// TIA Portal project "banc de percage" (V16)

(* hardware
DEVICE "Station S7-1200_1"  S7-1200 Station
   slot 0: "Châssis_0"  S7-1200 Rack  Rack  V1.0
   slot 1: "PLC_1"  CPU 1214C DC/DC/DC  6ES7 214-1AG31-0XB0  V3.0
*)

// ===== PLC "PLC_1"  CPU 1214C DC/DC/DC =====

VAR_GLOBAL   // PLC tag table "Table de variables standard"
   "S1" AT %I0.0 : Bool;
   "AU" AT %I0.1 : Bool;
   "DCA" AT %I0.2 : Bool;
   "FCA" AT %I0.3 : Bool;
   "DCB" AT %I0.4 : Bool;
   "FCB" AT %I0.5 : Bool;
   "FCC" AT %I0.6 : Bool;
   "PP" AT %I0.7 : Bool;
   "SWC" AT %I1.0 : Bool;
   "A12" AT %Q0.1 : Bool;
   "A14" AT %Q0.2 : Bool;
   "B12" AT %Q0.3 : Bool;
   "B14" AT %Q0.4 : Bool;
   "D12" AT %Q0.5 : Bool;
   "KM1" AT %Q0.6 : Bool;
   "H1" AT %Q0.7 : Bool;
   "H2" AT %Q1.0 : Bool;
   "Mot etape" AT %MW20 : Int;
   "Clock_Byte" AT %MB0 : Byte;
   "Clock_10Hz" AT %M0.0 : Bool;
   "Clock_5Hz" AT %M0.1 : Bool;
   "Clock_2.5Hz" AT %M0.2 : Bool;
   "Clock_2Hz" AT %M0.3 : Bool;
   "Clock_1.25Hz" AT %M0.4 : Bool;
   "Clock_1Hz" AT %M0.5 : Bool;
   "Clock_0.625Hz" AT %M0.6 : Bool;
   "Clock_0.5Hz" AT %M0.7 : Bool;
   "RAU" AT %I1.1 : Bool;
   "H3" AT %Q1.1 : Bool;
   "Reset" AT %E1.2 : Bool;
   "C12" AT %Q0.0 : Bool;
END_VAR

// folder: System blocks/Program resources

DATA_BLOCK "IEC_Timer_0_DB_1"   // DB2
{ S7_Optimized_Access := 'TRUE' }
AUTHOR : Simatic
FAMILY : IEC
NAME : IEC_TMR
VERSION : 1.0
// stored: InstanceOfName IEC_TIMER
"IEC_TIMER"
BEGIN
END_DATA_BLOCK

DATA_BLOCK "IEC_Timer_0_DB_2"   // DB3
{ S7_Optimized_Access := 'TRUE' }
AUTHOR : Simatic
FAMILY : IEC
NAME : IEC_TMR
VERSION : 1.0
// stored: InstanceOfName IEC_TIMER
"IEC_TIMER"
BEGIN
END_DATA_BLOCK

DATA_BLOCK "IEC_Timer_0_DB_3"   // DB4
{ S7_Optimized_Access := 'TRUE' }
AUTHOR : Simatic
FAMILY : IEC
NAME : IEC_TMR
VERSION : 1.0
// stored: InstanceOfName IEC_TIMER
"IEC_TIMER"
BEGIN
END_DATA_BLOCK

// folder: (top level)

FUNCTION "Transition" : Void   // FC1, LAD
{ S7_Optimized_Access := 'TRUE' }
VERSION : 0.1
   VAR_TEMP   // added for the SCL form of the ladder/FBD networks
      _w1 : Bool;
   END_VAR
BEGIN

REGION Network 1
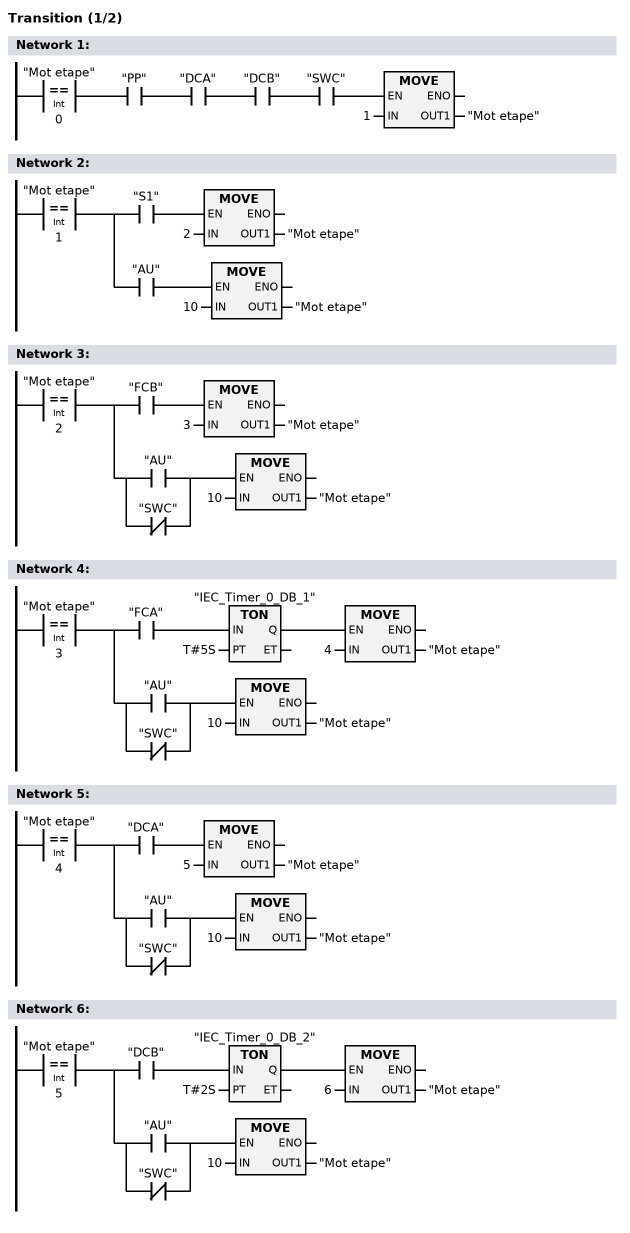
   RUNG wire#powerrail
      { S7_Templates := "SrcType := Int" } EQ_Contact(in1 := "Mot etape", in2 := 0)
      Contact( "PP" )
      Contact( "DCA" )
      Contact( "DCB" )
      Contact( "SWC" )
      { S7_GenerateENO := "TRUE" } Move(in := 1, out1 => "Mot etape")
   END_RUNG
   // the same network as SCL:
   IF ("Mot etape" = 0) AND "PP" AND "DCA" AND "DCB" AND "SWC" THEN "Mot etape" := 1; END_IF;
END_REGION

REGION Network 2
   RUNG wire#powerrail
      { S7_Templates := "SrcType := Int" } EQ_Contact(in1 := "Mot etape", in2 := 1)
      wire#w1
      Contact( "S1" )
      { S7_GenerateENO := "TRUE" } Move(in := 2, out1 => "Mot etape")
   END_RUNG
   RUNG wire#w1
      Contact( "AU" )
      { S7_GenerateENO := "TRUE" } Move(in := 10, out1 => "Mot etape")
   END_RUNG
   // the same network as SCL:
   #_w1 := "Mot etape" = 1;
   IF #_w1 AND "S1" THEN "Mot etape" := 2; END_IF;
   IF #_w1 AND "AU" THEN "Mot etape" := 10; END_IF;
END_REGION

REGION Network 3
   RUNG wire#powerrail
      { S7_Templates := "SrcType := Int" } EQ_Contact(in1 := "Mot etape", in2 := 2)
      wire#w1
      Contact( "FCB" )
      { S7_GenerateENO := "TRUE" } Move(in := 3, out1 => "Mot etape")
   END_RUNG
   RUNG wire#w1
      Contact( "AU" )
      wire#w2
      { S7_GenerateENO := "TRUE" } Move(in := 10, out1 => "Mot etape")
   END_RUNG
   RUNG wire#w1
      I_Contact( "SWC" )
   END_RUNG wire#w2
   // the same network as SCL:
   #_w1 := "Mot etape" = 2;
   IF #_w1 AND "FCB" THEN "Mot etape" := 3; END_IF;
   IF #_w1 AND ("AU" OR NOT "SWC") THEN "Mot etape" := 10; END_IF;
END_REGION

REGION Network 4
   #_w1 := "Mot etape" = 3;
   "IEC_Timer_0_DB_1".TON(IN := #_w1 AND "FCA", PT := T#5S);
   IF "IEC_Timer_0_DB_1".Q THEN "Mot etape" := 4; END_IF;
   IF #_w1 AND ("AU" OR NOT "SWC") THEN "Mot etape" := 10; END_IF;
END_REGION

REGION Network 5
   RUNG wire#powerrail
      { S7_Templates := "SrcType := Int" } EQ_Contact(in1 := "Mot etape", in2 := 4)
      wire#w1
      Contact( "DCA" )
      { S7_GenerateENO := "TRUE" } Move(in := 5, out1 => "Mot etape")
   END_RUNG
   RUNG wire#w1
      Contact( "AU" )
      wire#w2
      { S7_GenerateENO := "TRUE" } Move(in := 10, out1 => "Mot etape")
   END_RUNG
   RUNG wire#w1
      I_Contact( "SWC" )
   END_RUNG wire#w2
   // the same network as SCL:
   #_w1 := "Mot etape" = 4;
   IF #_w1 AND "DCA" THEN "Mot etape" := 5; END_IF;
   IF #_w1 AND ("AU" OR NOT "SWC") THEN "Mot etape" := 10; END_IF;
END_REGION

REGION Network 6
   #_w1 := "Mot etape" = 5;
   "IEC_Timer_0_DB_2".TON(IN := #_w1 AND "DCB", PT := T#2S);
   IF "IEC_Timer_0_DB_2".Q THEN "Mot etape" := 6; END_IF;
   IF #_w1 AND ("AU" OR NOT "SWC") THEN "Mot etape" := 10; END_IF;
END_REGION

REGION Network 7
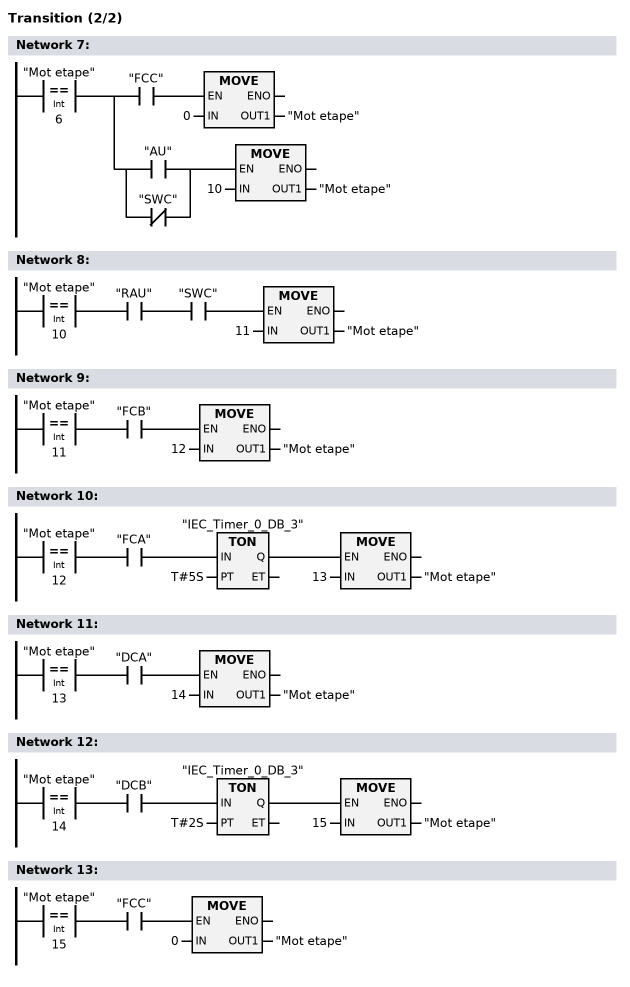
   RUNG wire#powerrail
      { S7_Templates := "SrcType := Int" } EQ_Contact(in1 := "Mot etape", in2 := 6)
      wire#w1
      Contact( "FCC" )
      { S7_GenerateENO := "TRUE" } Move(in := 0, out1 => "Mot etape")
   END_RUNG
   RUNG wire#w1
      Contact( "AU" )
      wire#w2
      { S7_GenerateENO := "TRUE" } Move(in := 10, out1 => "Mot etape")
   END_RUNG
   RUNG wire#w1
      I_Contact( "SWC" )
   END_RUNG wire#w2
   // the same network as SCL:
   #_w1 := "Mot etape" = 6;
   IF #_w1 AND "FCC" THEN "Mot etape" := 0; END_IF;
   IF #_w1 AND ("AU" OR NOT "SWC") THEN "Mot etape" := 10; END_IF;
END_REGION

REGION Network 8
   RUNG wire#powerrail
      { S7_Templates := "SrcType := Int" } EQ_Contact(in1 := "Mot etape", in2 := 10)
      Contact( "RAU" )
      Contact( "SWC" )
      { S7_GenerateENO := "TRUE" } Move(in := 11, out1 => "Mot etape")
   END_RUNG
   // the same network as SCL:
   IF ("Mot etape" = 10) AND "RAU" AND "SWC" THEN "Mot etape" := 11; END_IF;
END_REGION

REGION Network 9
   RUNG wire#powerrail
      { S7_Templates := "SrcType := Int" } EQ_Contact(in1 := "Mot etape", in2 := 11)
      Contact( "FCB" )
      { S7_GenerateENO := "TRUE" } Move(in := 12, out1 => "Mot etape")
   END_RUNG
   // the same network as SCL:
   IF ("Mot etape" = 11) AND "FCB" THEN "Mot etape" := 12; END_IF;
END_REGION

REGION Network 10
   "IEC_Timer_0_DB_3".TON(IN := ("Mot etape" = 12) AND "FCA", PT := T#5S);
   IF "IEC_Timer_0_DB_3".Q THEN "Mot etape" := 13; END_IF;
END_REGION

REGION Network 11
   RUNG wire#powerrail
      { S7_Templates := "SrcType := Int" } EQ_Contact(in1 := "Mot etape", in2 := 13)
      Contact( "DCA" )
      { S7_GenerateENO := "TRUE" } Move(in := 14, out1 => "Mot etape")
   END_RUNG
   // the same network as SCL:
   IF ("Mot etape" = 13) AND "DCA" THEN "Mot etape" := 14; END_IF;
END_REGION

REGION Network 12
   "IEC_Timer_0_DB_3".TON(IN := ("Mot etape" = 14) AND "DCB", PT := T#2S);
   IF "IEC_Timer_0_DB_3".Q THEN "Mot etape" := 15; END_IF;
END_REGION

REGION Network 13
   RUNG wire#powerrail
      { S7_Templates := "SrcType := Int" } EQ_Contact(in1 := "Mot etape", in2 := 15)
      Contact( "FCC" )
      { S7_GenerateENO := "TRUE" } Move(in := 0, out1 => "Mot etape")
   END_RUNG
   // the same network as SCL:
   IF ("Mot etape" = 15) AND "FCC" THEN "Mot etape" := 0; END_IF;
END_REGION
END_FUNCTION

FUNCTION "Sortie" : Void   // FC2, LAD
{ S7_Optimized_Access := 'TRUE' }
VERSION : 0.1
BEGIN

REGION Network 1
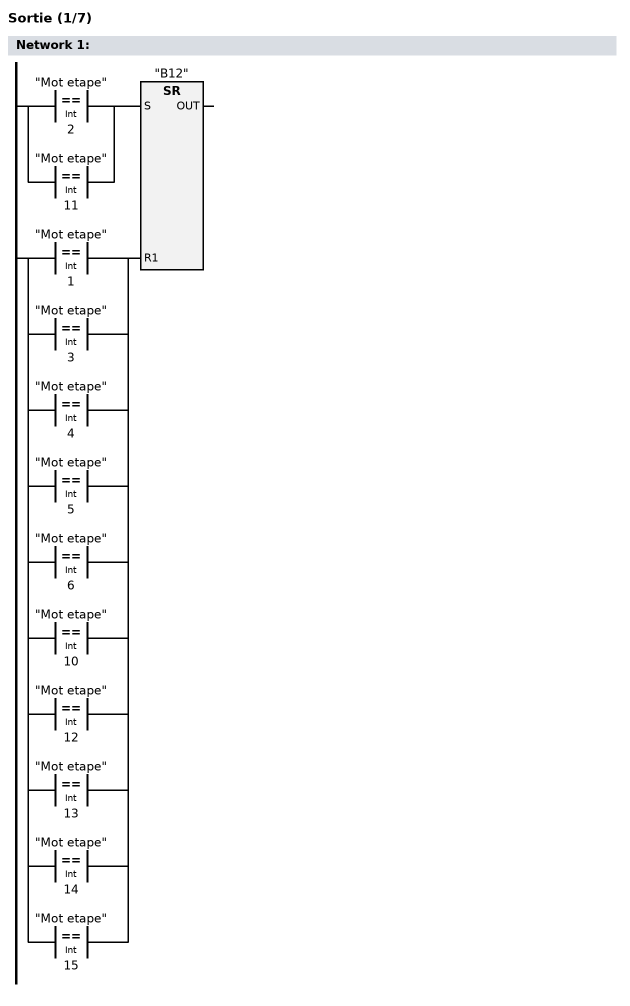
   RUNG wire#powerrail
      { S7_Templates := "SrcType := Int" } EQ_Contact(in1 := "Mot etape", in2 := 2)
      wire#w1
      S_SR(operand := "B12", r1 := wire#w2)
   END_RUNG
   RUNG wire#powerrail
      { S7_Templates := "SrcType := Int" } EQ_Contact(in1 := "Mot etape", in2 := 11)
   END_RUNG wire#w1
   RUNG wire#powerrail
      { S7_Templates := "SrcType := Int" } EQ_Contact(in1 := "Mot etape", in2 := 1)
   END_RUNG wire#w2
   RUNG wire#powerrail
      { S7_Templates := "SrcType := Int" } EQ_Contact(in1 := "Mot etape", in2 := 3)
   END_RUNG wire#w2
   RUNG wire#powerrail
      { S7_Templates := "SrcType := Int" } EQ_Contact(in1 := "Mot etape", in2 := 4)
   END_RUNG wire#w2
   RUNG wire#powerrail
      { S7_Templates := "SrcType := Int" } EQ_Contact(in1 := "Mot etape", in2 := 5)
   END_RUNG wire#w2
   RUNG wire#powerrail
      { S7_Templates := "SrcType := Int" } EQ_Contact(in1 := "Mot etape", in2 := 6)
   END_RUNG wire#w2
   RUNG wire#powerrail
      { S7_Templates := "SrcType := Int" } EQ_Contact(in1 := "Mot etape", in2 := 10)
   END_RUNG wire#w2
   RUNG wire#powerrail
      { S7_Templates := "SrcType := Int" } EQ_Contact(in1 := "Mot etape", in2 := 12)
   END_RUNG wire#w2
   RUNG wire#powerrail
      { S7_Templates := "SrcType := Int" } EQ_Contact(in1 := "Mot etape", in2 := 13)
   END_RUNG wire#w2
   RUNG wire#powerrail
      { S7_Templates := "SrcType := Int" } EQ_Contact(in1 := "Mot etape", in2 := 14)
   END_RUNG wire#w2
   RUNG wire#powerrail
      { S7_Templates := "SrcType := Int" } EQ_Contact(in1 := "Mot etape", in2 := 15)
   END_RUNG wire#w2
   // the same network as SCL:
   IF ("Mot etape" = 2) OR ("Mot etape" = 11) THEN
       "B12" := TRUE;   // SR flip-flop
   END_IF;
   IF ("Mot etape" = 1) OR ("Mot etape" = 3) OR ("Mot etape" = 4) OR ("Mot etape" = 5) OR ("Mot etape" = 6) OR ("Mot etape" = 10) OR ("Mot etape" = 12) OR ("Mot etape" = 13) OR ("Mot etape" = 14) OR ("Mot etape" = 15) THEN
       "B12" := FALSE;
   END_IF;
END_REGION

REGION Network 2
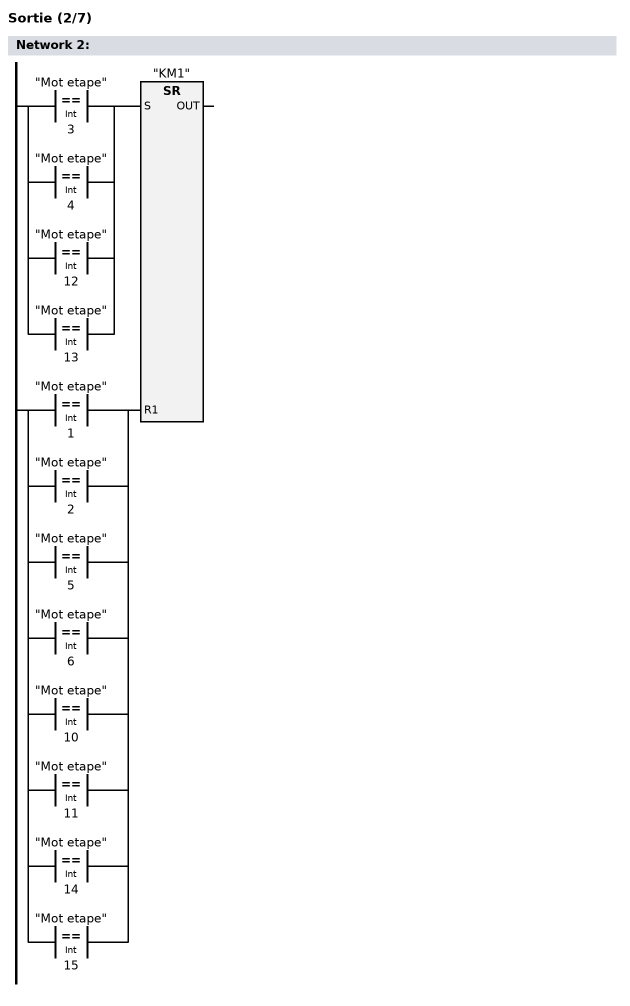
   RUNG wire#powerrail
      { S7_Templates := "SrcType := Int" } EQ_Contact(in1 := "Mot etape", in2 := 3)
      wire#w1
      S_SR(operand := "KM1", r1 := wire#w2)
   END_RUNG
   RUNG wire#powerrail
      { S7_Templates := "SrcType := Int" } EQ_Contact(in1 := "Mot etape", in2 := 4)
   END_RUNG wire#w1
   RUNG wire#powerrail
      { S7_Templates := "SrcType := Int" } EQ_Contact(in1 := "Mot etape", in2 := 12)
   END_RUNG wire#w1
   RUNG wire#powerrail
      { S7_Templates := "SrcType := Int" } EQ_Contact(in1 := "Mot etape", in2 := 13)
   END_RUNG wire#w1
   RUNG wire#powerrail
      { S7_Templates := "SrcType := Int" } EQ_Contact(in1 := "Mot etape", in2 := 1)
   END_RUNG wire#w2
   RUNG wire#powerrail
      { S7_Templates := "SrcType := Int" } EQ_Contact(in1 := "Mot etape", in2 := 2)
   END_RUNG wire#w2
   RUNG wire#powerrail
      { S7_Templates := "SrcType := Int" } EQ_Contact(in1 := "Mot etape", in2 := 5)
   END_RUNG wire#w2
   RUNG wire#powerrail
      { S7_Templates := "SrcType := Int" } EQ_Contact(in1 := "Mot etape", in2 := 6)
   END_RUNG wire#w2
   RUNG wire#powerrail
      { S7_Templates := "SrcType := Int" } EQ_Contact(in1 := "Mot etape", in2 := 10)
   END_RUNG wire#w2
   RUNG wire#powerrail
      { S7_Templates := "SrcType := Int" } EQ_Contact(in1 := "Mot etape", in2 := 11)
   END_RUNG wire#w2
   RUNG wire#powerrail
      { S7_Templates := "SrcType := Int" } EQ_Contact(in1 := "Mot etape", in2 := 14)
   END_RUNG wire#w2
   RUNG wire#powerrail
      { S7_Templates := "SrcType := Int" } EQ_Contact(in1 := "Mot etape", in2 := 15)
   END_RUNG wire#w2
   // the same network as SCL:
   IF ("Mot etape" = 3) OR ("Mot etape" = 4) OR ("Mot etape" = 12) OR ("Mot etape" = 13) THEN
       "KM1" := TRUE;   // SR flip-flop
   END_IF;
   IF ("Mot etape" = 1) OR ("Mot etape" = 2) OR ("Mot etape" = 5) OR ("Mot etape" = 6) OR ("Mot etape" = 10) OR ("Mot etape" = 11) OR ("Mot etape" = 14) OR ("Mot etape" = 15) THEN
       "KM1" := FALSE;
   END_IF;
END_REGION

REGION Network 3
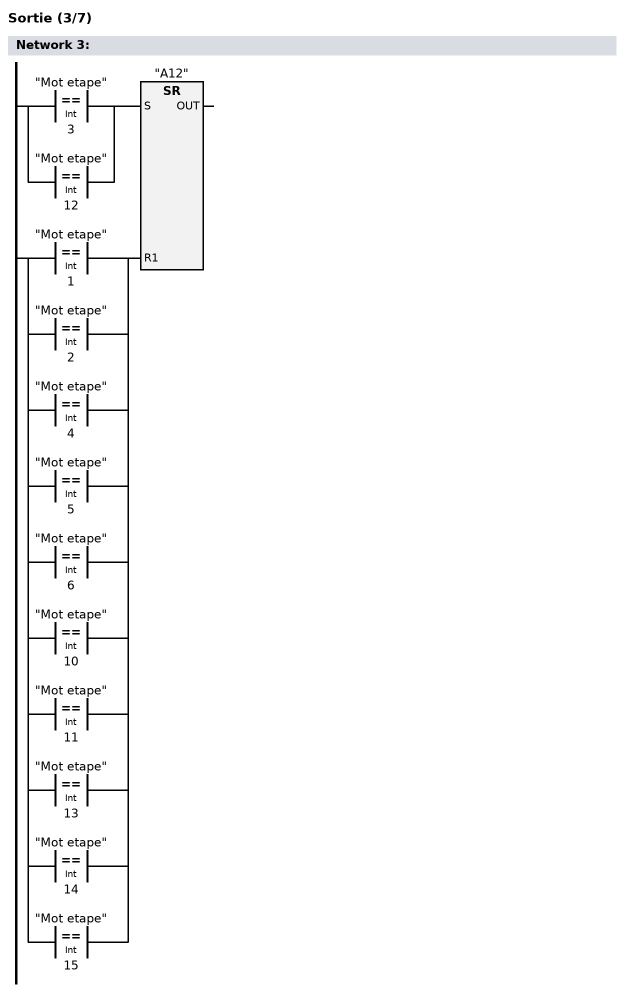
   RUNG wire#powerrail
      { S7_Templates := "SrcType := Int" } EQ_Contact(in1 := "Mot etape", in2 := 3)
      wire#w1
      S_SR(operand := "A12", r1 := wire#w2)
   END_RUNG
   RUNG wire#powerrail
      { S7_Templates := "SrcType := Int" } EQ_Contact(in1 := "Mot etape", in2 := 12)
   END_RUNG wire#w1
   RUNG wire#powerrail
      { S7_Templates := "SrcType := Int" } EQ_Contact(in1 := "Mot etape", in2 := 1)
   END_RUNG wire#w2
   RUNG wire#powerrail
      { S7_Templates := "SrcType := Int" } EQ_Contact(in1 := "Mot etape", in2 := 2)
   END_RUNG wire#w2
   RUNG wire#powerrail
      { S7_Templates := "SrcType := Int" } EQ_Contact(in1 := "Mot etape", in2 := 4)
   END_RUNG wire#w2
   RUNG wire#powerrail
      { S7_Templates := "SrcType := Int" } EQ_Contact(in1 := "Mot etape", in2 := 5)
   END_RUNG wire#w2
   RUNG wire#powerrail
      { S7_Templates := "SrcType := Int" } EQ_Contact(in1 := "Mot etape", in2 := 6)
   END_RUNG wire#w2
   RUNG wire#powerrail
      { S7_Templates := "SrcType := Int" } EQ_Contact(in1 := "Mot etape", in2 := 10)
   END_RUNG wire#w2
   RUNG wire#powerrail
      { S7_Templates := "SrcType := Int" } EQ_Contact(in1 := "Mot etape", in2 := 11)
   END_RUNG wire#w2
   RUNG wire#powerrail
      { S7_Templates := "SrcType := Int" } EQ_Contact(in1 := "Mot etape", in2 := 13)
   END_RUNG wire#w2
   RUNG wire#powerrail
      { S7_Templates := "SrcType := Int" } EQ_Contact(in1 := "Mot etape", in2 := 14)
   END_RUNG wire#w2
   RUNG wire#powerrail
      { S7_Templates := "SrcType := Int" } EQ_Contact(in1 := "Mot etape", in2 := 15)
   END_RUNG wire#w2
   // the same network as SCL:
   IF ("Mot etape" = 3) OR ("Mot etape" = 12) THEN
       "A12" := TRUE;   // SR flip-flop
   END_IF;
   IF ("Mot etape" = 1) OR ("Mot etape" = 2) OR ("Mot etape" = 4) OR ("Mot etape" = 5) OR ("Mot etape" = 6) OR ("Mot etape" = 10) OR ("Mot etape" = 11) OR ("Mot etape" = 13) OR ("Mot etape" = 14) OR ("Mot etape" = 15) THEN
       "A12" := FALSE;
   END_IF;
END_REGION

REGION Network 4
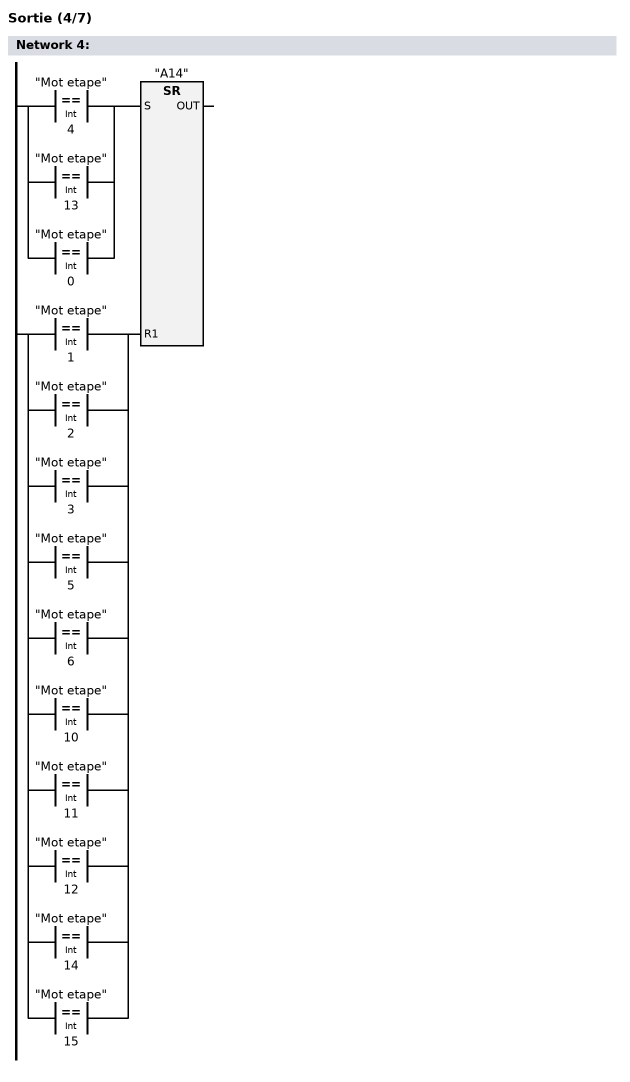
   RUNG wire#powerrail
      { S7_Templates := "SrcType := Int" } EQ_Contact(in1 := "Mot etape", in2 := 4)
      wire#w1
      S_SR(operand := "A14", r1 := wire#w2)
   END_RUNG
   RUNG wire#powerrail
      { S7_Templates := "SrcType := Int" } EQ_Contact(in1 := "Mot etape", in2 := 13)
   END_RUNG wire#w1
   RUNG wire#powerrail
      { S7_Templates := "SrcType := Int" } EQ_Contact(in1 := "Mot etape", in2 := 0)
   END_RUNG wire#w1
   RUNG wire#powerrail
      { S7_Templates := "SrcType := Int" } EQ_Contact(in1 := "Mot etape", in2 := 1)
   END_RUNG wire#w2
   RUNG wire#powerrail
      { S7_Templates := "SrcType := Int" } EQ_Contact(in1 := "Mot etape", in2 := 2)
   END_RUNG wire#w2
   RUNG wire#powerrail
      { S7_Templates := "SrcType := Int" } EQ_Contact(in1 := "Mot etape", in2 := 3)
   END_RUNG wire#w2
   RUNG wire#powerrail
      { S7_Templates := "SrcType := Int" } EQ_Contact(in1 := "Mot etape", in2 := 5)
   END_RUNG wire#w2
   RUNG wire#powerrail
      { S7_Templates := "SrcType := Int" } EQ_Contact(in1 := "Mot etape", in2 := 6)
   END_RUNG wire#w2
   RUNG wire#powerrail
      { S7_Templates := "SrcType := Int" } EQ_Contact(in1 := "Mot etape", in2 := 10)
   END_RUNG wire#w2
   RUNG wire#powerrail
      { S7_Templates := "SrcType := Int" } EQ_Contact(in1 := "Mot etape", in2 := 11)
   END_RUNG wire#w2
   RUNG wire#powerrail
      { S7_Templates := "SrcType := Int" } EQ_Contact(in1 := "Mot etape", in2 := 12)
   END_RUNG wire#w2
   RUNG wire#powerrail
      { S7_Templates := "SrcType := Int" } EQ_Contact(in1 := "Mot etape", in2 := 14)
   END_RUNG wire#w2
   RUNG wire#powerrail
      { S7_Templates := "SrcType := Int" } EQ_Contact(in1 := "Mot etape", in2 := 15)
   END_RUNG wire#w2
   // the same network as SCL:
   IF ("Mot etape" = 4) OR ("Mot etape" = 13) OR ("Mot etape" = 0) THEN
       "A14" := TRUE;   // SR flip-flop
   END_IF;
   IF ("Mot etape" = 1) OR ("Mot etape" = 2) OR ("Mot etape" = 3) OR ("Mot etape" = 5) OR ("Mot etape" = 6) OR ("Mot etape" = 10) OR ("Mot etape" = 11) OR ("Mot etape" = 12) OR ("Mot etape" = 14) OR ("Mot etape" = 15) THEN
       "A14" := FALSE;
   END_IF;
END_REGION

REGION Network 5
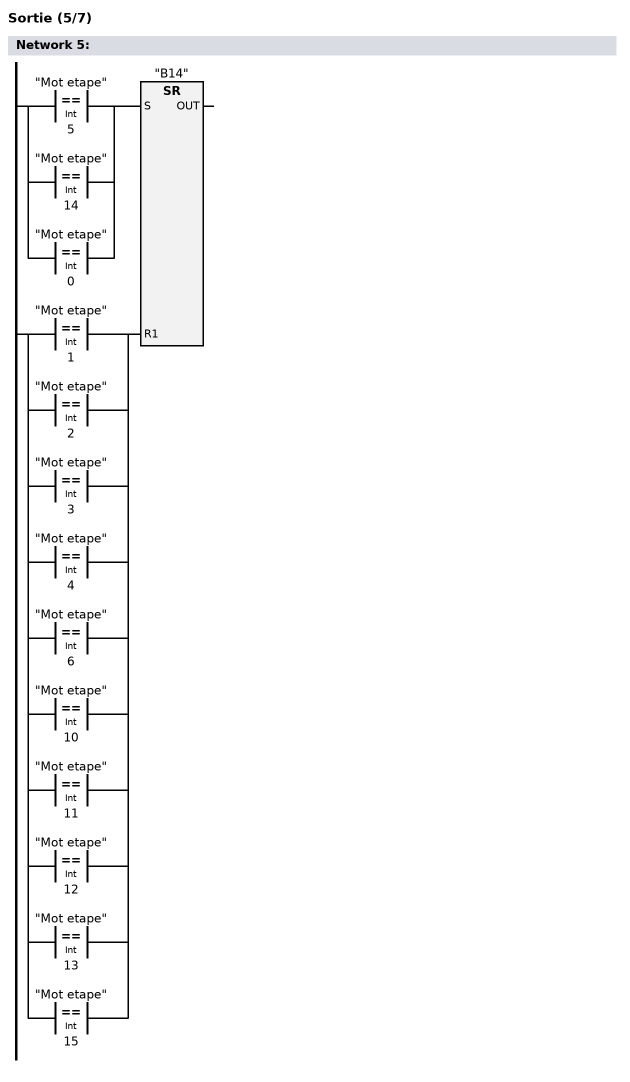
   RUNG wire#powerrail
      { S7_Templates := "SrcType := Int" } EQ_Contact(in1 := "Mot etape", in2 := 5)
      wire#w1
      S_SR(operand := "B14", r1 := wire#w2)
   END_RUNG
   RUNG wire#powerrail
      { S7_Templates := "SrcType := Int" } EQ_Contact(in1 := "Mot etape", in2 := 14)
   END_RUNG wire#w1
   RUNG wire#powerrail
      { S7_Templates := "SrcType := Int" } EQ_Contact(in1 := "Mot etape", in2 := 0)
   END_RUNG wire#w1
   RUNG wire#powerrail
      { S7_Templates := "SrcType := Int" } EQ_Contact(in1 := "Mot etape", in2 := 1)
   END_RUNG wire#w2
   RUNG wire#powerrail
      { S7_Templates := "SrcType := Int" } EQ_Contact(in1 := "Mot etape", in2 := 2)
   END_RUNG wire#w2
   RUNG wire#powerrail
      { S7_Templates := "SrcType := Int" } EQ_Contact(in1 := "Mot etape", in2 := 3)
   END_RUNG wire#w2
   RUNG wire#powerrail
      { S7_Templates := "SrcType := Int" } EQ_Contact(in1 := "Mot etape", in2 := 4)
   END_RUNG wire#w2
   RUNG wire#powerrail
      { S7_Templates := "SrcType := Int" } EQ_Contact(in1 := "Mot etape", in2 := 6)
   END_RUNG wire#w2
   RUNG wire#powerrail
      { S7_Templates := "SrcType := Int" } EQ_Contact(in1 := "Mot etape", in2 := 10)
   END_RUNG wire#w2
   RUNG wire#powerrail
      { S7_Templates := "SrcType := Int" } EQ_Contact(in1 := "Mot etape", in2 := 11)
   END_RUNG wire#w2
   RUNG wire#powerrail
      { S7_Templates := "SrcType := Int" } EQ_Contact(in1 := "Mot etape", in2 := 12)
   END_RUNG wire#w2
   RUNG wire#powerrail
      { S7_Templates := "SrcType := Int" } EQ_Contact(in1 := "Mot etape", in2 := 13)
   END_RUNG wire#w2
   RUNG wire#powerrail
      { S7_Templates := "SrcType := Int" } EQ_Contact(in1 := "Mot etape", in2 := 15)
   END_RUNG wire#w2
   // the same network as SCL:
   IF ("Mot etape" = 5) OR ("Mot etape" = 14) OR ("Mot etape" = 0) THEN
       "B14" := TRUE;   // SR flip-flop
   END_IF;
   IF ("Mot etape" = 1) OR ("Mot etape" = 2) OR ("Mot etape" = 3) OR ("Mot etape" = 4) OR ("Mot etape" = 6) OR ("Mot etape" = 10) OR ("Mot etape" = 11) OR ("Mot etape" = 12) OR ("Mot etape" = 13) OR ("Mot etape" = 15) THEN
       "B14" := FALSE;
   END_IF;
END_REGION

REGION Network 6
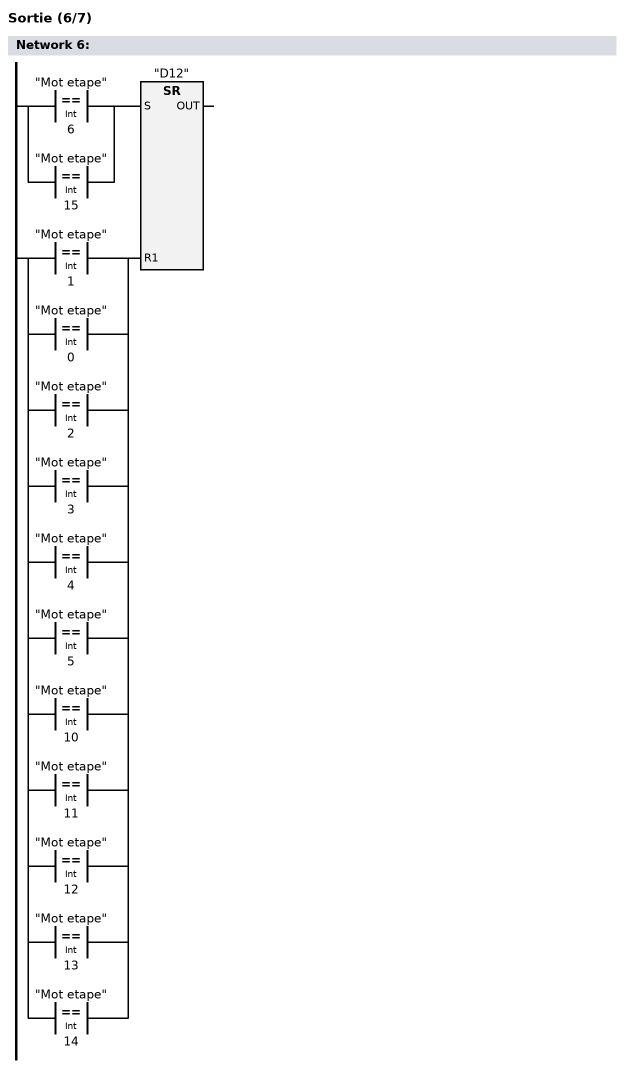
   RUNG wire#powerrail
      { S7_Templates := "SrcType := Int" } EQ_Contact(in1 := "Mot etape", in2 := 6)
      wire#w1
      S_SR(operand := "D12", r1 := wire#w2)
   END_RUNG
   RUNG wire#powerrail
      { S7_Templates := "SrcType := Int" } EQ_Contact(in1 := "Mot etape", in2 := 15)
   END_RUNG wire#w1
   RUNG wire#powerrail
      { S7_Templates := "SrcType := Int" } EQ_Contact(in1 := "Mot etape", in2 := 1)
   END_RUNG wire#w2
   RUNG wire#powerrail
      { S7_Templates := "SrcType := Int" } EQ_Contact(in1 := "Mot etape", in2 := 0)
   END_RUNG wire#w2
   RUNG wire#powerrail
      { S7_Templates := "SrcType := Int" } EQ_Contact(in1 := "Mot etape", in2 := 2)
   END_RUNG wire#w2
   RUNG wire#powerrail
      { S7_Templates := "SrcType := Int" } EQ_Contact(in1 := "Mot etape", in2 := 3)
   END_RUNG wire#w2
   RUNG wire#powerrail
      { S7_Templates := "SrcType := Int" } EQ_Contact(in1 := "Mot etape", in2 := 4)
   END_RUNG wire#w2
   RUNG wire#powerrail
      { S7_Templates := "SrcType := Int" } EQ_Contact(in1 := "Mot etape", in2 := 5)
   END_RUNG wire#w2
   RUNG wire#powerrail
      { S7_Templates := "SrcType := Int" } EQ_Contact(in1 := "Mot etape", in2 := 10)
   END_RUNG wire#w2
   RUNG wire#powerrail
      { S7_Templates := "SrcType := Int" } EQ_Contact(in1 := "Mot etape", in2 := 11)
   END_RUNG wire#w2
   RUNG wire#powerrail
      { S7_Templates := "SrcType := Int" } EQ_Contact(in1 := "Mot etape", in2 := 12)
   END_RUNG wire#w2
   RUNG wire#powerrail
      { S7_Templates := "SrcType := Int" } EQ_Contact(in1 := "Mot etape", in2 := 13)
   END_RUNG wire#w2
   RUNG wire#powerrail
      { S7_Templates := "SrcType := Int" } EQ_Contact(in1 := "Mot etape", in2 := 14)
   END_RUNG wire#w2
   // the same network as SCL:
   IF ("Mot etape" = 6) OR ("Mot etape" = 15) THEN
       "D12" := TRUE;   // SR flip-flop
   END_IF;
   IF ("Mot etape" = 1) OR ("Mot etape" = 0) OR ("Mot etape" = 2) OR ("Mot etape" = 3) OR ("Mot etape" = 4) OR ("Mot etape" = 5) OR ("Mot etape" = 10) OR ("Mot etape" = 11) OR ("Mot etape" = 12) OR ("Mot etape" = 13) OR ("Mot etape" = 14) THEN
       "D12" := FALSE;
   END_IF;
END_REGION

REGION Network 7
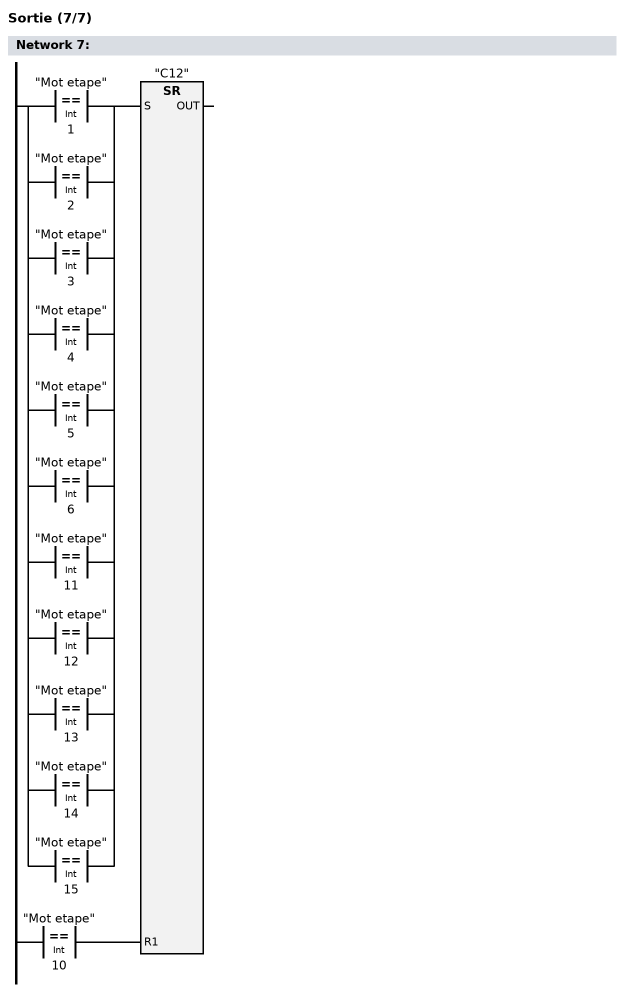
   RUNG wire#powerrail
      { S7_Templates := "SrcType := Int" } EQ_Contact(in1 := "Mot etape", in2 := 1)
      wire#w1
      S_SR(operand := "C12", r1 := wire#w2)
   END_RUNG
   RUNG wire#powerrail
      { S7_Templates := "SrcType := Int" } EQ_Contact(in1 := "Mot etape", in2 := 2)
   END_RUNG wire#w1
   RUNG wire#powerrail
      { S7_Templates := "SrcType := Int" } EQ_Contact(in1 := "Mot etape", in2 := 3)
   END_RUNG wire#w1
   RUNG wire#powerrail
      { S7_Templates := "SrcType := Int" } EQ_Contact(in1 := "Mot etape", in2 := 4)
   END_RUNG wire#w1
   RUNG wire#powerrail
      { S7_Templates := "SrcType := Int" } EQ_Contact(in1 := "Mot etape", in2 := 5)
   END_RUNG wire#w1
   RUNG wire#powerrail
      { S7_Templates := "SrcType := Int" } EQ_Contact(in1 := "Mot etape", in2 := 6)
   END_RUNG wire#w1
   RUNG wire#powerrail
      { S7_Templates := "SrcType := Int" } EQ_Contact(in1 := "Mot etape", in2 := 11)
   END_RUNG wire#w1
   RUNG wire#powerrail
      { S7_Templates := "SrcType := Int" } EQ_Contact(in1 := "Mot etape", in2 := 12)
   END_RUNG wire#w1
   RUNG wire#powerrail
      { S7_Templates := "SrcType := Int" } EQ_Contact(in1 := "Mot etape", in2 := 13)
   END_RUNG wire#w1
   RUNG wire#powerrail
      { S7_Templates := "SrcType := Int" } EQ_Contact(in1 := "Mot etape", in2 := 14)
   END_RUNG wire#w1
   RUNG wire#powerrail
      { S7_Templates := "SrcType := Int" } EQ_Contact(in1 := "Mot etape", in2 := 15)
   END_RUNG wire#w1
   RUNG wire#powerrail
      { S7_Templates := "SrcType := Int" } EQ_Contact(in1 := "Mot etape", in2 := 10)
   END_RUNG wire#w2
   // the same network as SCL:
   IF ("Mot etape" = 1) OR ("Mot etape" = 2) OR ("Mot etape" = 3) OR ("Mot etape" = 4) OR ("Mot etape" = 5) OR ("Mot etape" = 6) OR ("Mot etape" = 11) OR ("Mot etape" = 12) OR ("Mot etape" = 13) OR ("Mot etape" = 14) OR ("Mot etape" = 15) THEN
       "C12" := TRUE;   // SR flip-flop
   END_IF;
   IF "Mot etape" = 10 THEN "C12" := FALSE; END_IF;
END_REGION
END_FUNCTION

FUNCTION "Signalisation" : Void   // FC3, LAD
{ S7_Optimized_Access := 'TRUE' }
VERSION : 0.1
BEGIN

REGION Network 1
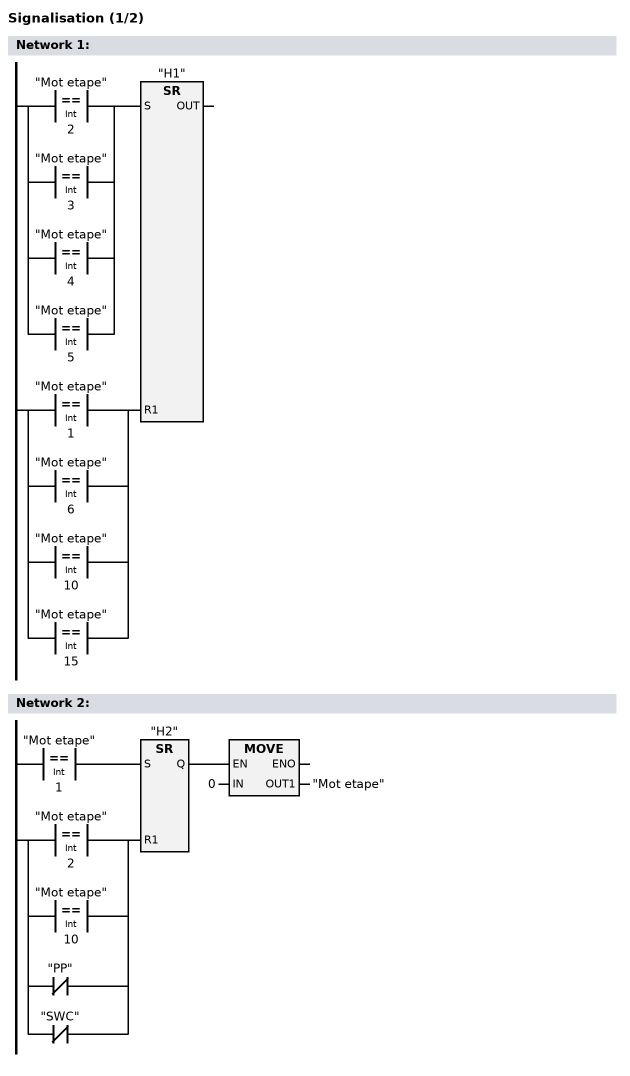
   RUNG wire#powerrail
      { S7_Templates := "SrcType := Int" } EQ_Contact(in1 := "Mot etape", in2 := 2)
      wire#w1
      S_SR(operand := "H1", r1 := wire#w2)
   END_RUNG
   RUNG wire#powerrail
      { S7_Templates := "SrcType := Int" } EQ_Contact(in1 := "Mot etape", in2 := 3)
   END_RUNG wire#w1
   RUNG wire#powerrail
      { S7_Templates := "SrcType := Int" } EQ_Contact(in1 := "Mot etape", in2 := 4)
   END_RUNG wire#w1
   RUNG wire#powerrail
      { S7_Templates := "SrcType := Int" } EQ_Contact(in1 := "Mot etape", in2 := 5)
   END_RUNG wire#w1
   RUNG wire#powerrail
      { S7_Templates := "SrcType := Int" } EQ_Contact(in1 := "Mot etape", in2 := 1)
   END_RUNG wire#w2
   RUNG wire#powerrail
      { S7_Templates := "SrcType := Int" } EQ_Contact(in1 := "Mot etape", in2 := 6)
   END_RUNG wire#w2
   RUNG wire#powerrail
      { S7_Templates := "SrcType := Int" } EQ_Contact(in1 := "Mot etape", in2 := 10)
   END_RUNG wire#w2
   RUNG wire#powerrail
      { S7_Templates := "SrcType := Int" } EQ_Contact(in1 := "Mot etape", in2 := 15)
   END_RUNG wire#w2
   // the same network as SCL:
   IF ("Mot etape" = 2) OR ("Mot etape" = 3) OR ("Mot etape" = 4) OR ("Mot etape" = 5) THEN
       "H1" := TRUE;   // SR flip-flop
   END_IF;
   IF ("Mot etape" = 1) OR ("Mot etape" = 6) OR ("Mot etape" = 10) OR ("Mot etape" = 15) THEN
       "H1" := FALSE;
   END_IF;
END_REGION

REGION Network 2
   RUNG wire#powerrail
      { S7_Templates := "SrcType := Int" } EQ_Contact(in1 := "Mot etape", in2 := 1)
      S_SR(operand := "H2", r1 := wire#w1)
      { S7_GenerateENO := "TRUE" } Move(in := 0, out1 => "Mot etape")
   END_RUNG
   RUNG wire#powerrail
      { S7_Templates := "SrcType := Int" } EQ_Contact(in1 := "Mot etape", in2 := 2)
   END_RUNG wire#w1
   RUNG wire#powerrail
      { S7_Templates := "SrcType := Int" } EQ_Contact(in1 := "Mot etape", in2 := 10)
   END_RUNG wire#w1
   RUNG wire#powerrail
      I_Contact( "PP" )
   END_RUNG wire#w1
   RUNG wire#powerrail
      I_Contact( "SWC" )
   END_RUNG wire#w1
   // the same network as SCL:
   IF "Mot etape" = 1 THEN
       "H2" := TRUE;   // SR flip-flop
   END_IF;
   IF ("Mot etape" = 2) OR ("Mot etape" = 10) OR NOT "PP" OR NOT "SWC" THEN "H2" := FALSE; END_IF;
   IF "H2" THEN "Mot etape" := 0; END_IF;
END_REGION

REGION Network 3
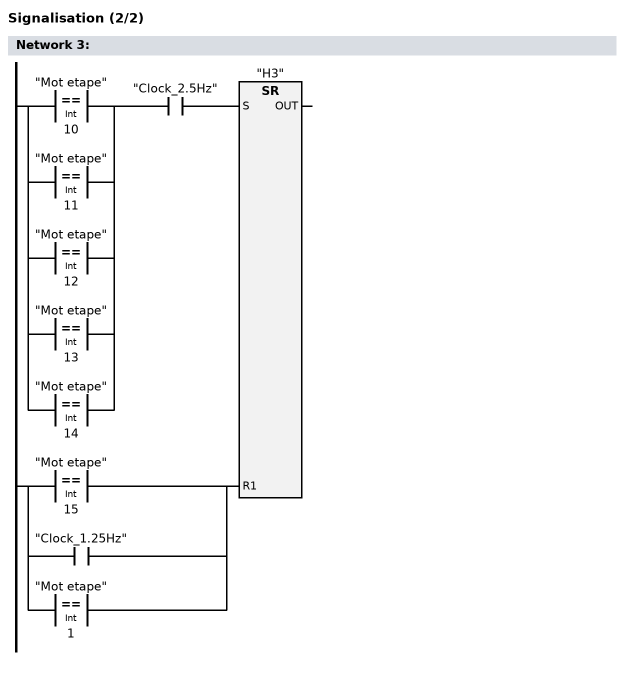
   RUNG wire#powerrail
      { S7_Templates := "SrcType := Int" } EQ_Contact(in1 := "Mot etape", in2 := 10)
      wire#w1
      Contact( "Clock_2.5Hz" )
      S_SR(operand := "H3", r1 := wire#w2)
   END_RUNG
   RUNG wire#powerrail
      { S7_Templates := "SrcType := Int" } EQ_Contact(in1 := "Mot etape", in2 := 11)
   END_RUNG wire#w1
   RUNG wire#powerrail
      { S7_Templates := "SrcType := Int" } EQ_Contact(in1 := "Mot etape", in2 := 12)
   END_RUNG wire#w1
   RUNG wire#powerrail
      { S7_Templates := "SrcType := Int" } EQ_Contact(in1 := "Mot etape", in2 := 13)
   END_RUNG wire#w1
   RUNG wire#powerrail
      { S7_Templates := "SrcType := Int" } EQ_Contact(in1 := "Mot etape", in2 := 14)
   END_RUNG wire#w1
   RUNG wire#powerrail
      { S7_Templates := "SrcType := Int" } EQ_Contact(in1 := "Mot etape", in2 := 15)
   END_RUNG wire#w2
   RUNG wire#powerrail
      Contact( "Clock_1.25Hz" )
   END_RUNG wire#w2
   RUNG wire#powerrail
      { S7_Templates := "SrcType := Int" } EQ_Contact(in1 := "Mot etape", in2 := 1)
   END_RUNG wire#w2
   // the same network as SCL:
   IF (("Mot etape" = 10) OR ("Mot etape" = 11) OR ("Mot etape" = 12) OR ("Mot etape" = 13) OR ("Mot etape" = 14)) AND "Clock_2.5Hz" THEN
       "H3" := TRUE;   // SR flip-flop
   END_IF;
   IF ("Mot etape" = 15) OR "Clock_1.25Hz" OR ("Mot etape" = 1) THEN "H3" := FALSE; END_IF;
END_REGION
END_FUNCTION

ORGANIZATION_BLOCK "Main"   // OB1, LAD, ProgramCycle
TITLE = "Main Program Sweep (Cycle)"
{ S7_Optimized_Access := 'TRUE' }
VERSION : 0.1
BEGIN

REGION Network 1
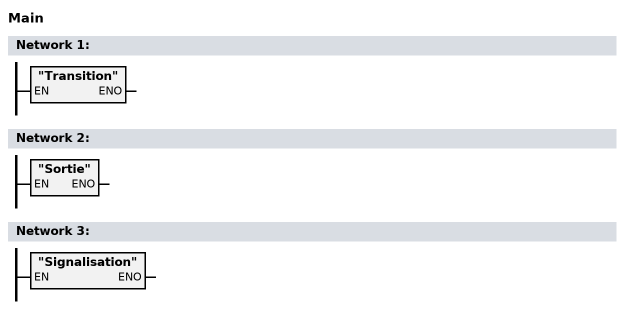
   RUNG wire#powerrail
      "Transition"()
   END_RUNG
   // the same network as SCL:
   "Transition"();
END_REGION

REGION Network 2
   RUNG wire#powerrail
      "Sortie"()
   END_RUNG
   // the same network as SCL:
   "Sortie"();
END_REGION

REGION Network 3
   RUNG wire#powerrail
      "Signalisation"()
   END_RUNG
   // the same network as SCL:
   "Signalisation"();
END_REGION
END_ORGANIZATION_BLOCK

ORGANIZATION_BLOCK "Startup"   // OB100, LAD, Startup
TITLE = "Complete Restart"
{ S7_Optimized_Access := 'TRUE' }
VERSION : 0.1
   VAR_INPUT
      LostRetentive : Bool;   // True if retentive data are lost
      LostRTC : Bool;   // True if date and time are lost
   END_VAR
BEGIN

REGION Network 1
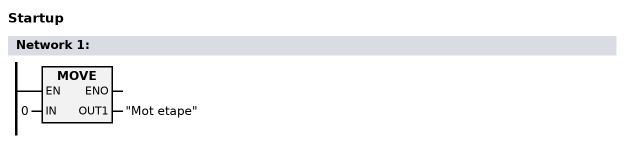
   RUNG wire#powerrail
      { S7_GenerateENO := "TRUE" } Move(in := 0, out1 => "Mot etape")
   END_RUNG
   // the same network as SCL:
   "Mot etape" := 0;
END_REGION
END_ORGANIZATION_BLOCK